(* CoDeSys 2.3.9.50 project: 4G.pr6 *)
(* Libraries: STANDARD.LB6 5.6.98 12:03:02 *)

(* POU MAIN, LD *)
PROGRAM MAIN
VAR
	Parts AT %IX0.0: BOOL;
	C1: CTU;
	Conveyer1 AT %QX0.0: BOOL;
	A AT %IX0.7: BOOL;
	C2: CTU;
	Reset AT %IX0.7: BOOL;
END_VAR
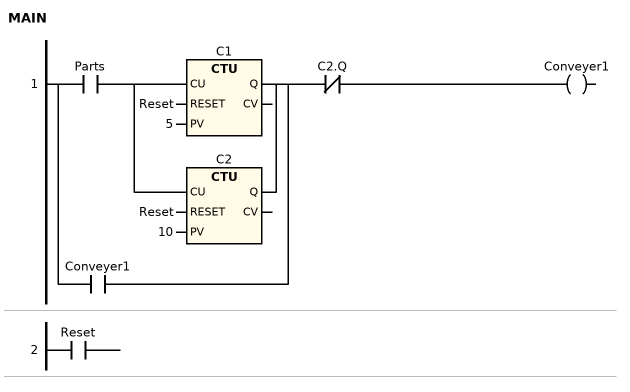
_LD_ (* Ladder Diagram *)
NETWORK 1
	{ [Parts] - { C1:CTU(CU: *, RESET: Reset, PV: 5) | C2:CTU(CU: *, RESET: Reset, PV: 10) } | [Conveyer1] } - [/C2.Q] --- (Conveyer1)
NETWORK 2
	[Reset]
_END_LD_
(* the same logic as Structured Text *)
(* Network 1 *)
C1(CU := Parts, RESET := Reset, PV := 5);
C2(CU := Parts, RESET := Reset, PV := 10);
Conveyer1 := ((C1.Q OR C2.Q) OR Conveyer1) AND NOT C2.Q;
(* Network 2 *)
END_PROGRAM
